{attribute 'linkalways'} 
{attribute 'no_explicit_call' := 'This FB is a CLASS and must be accessed using methods or properties'}
{attribute 'enable_dynamic_creation'}
FUNCTION_BLOCK _ETcVnSta EXTENDS EnumDatatypeBase
VAR
	localData : ETcVnSta;
	activeData : REFERENCE TO ETcVnSta;
	enumBaseDatatype : _UDINT(localData);
END_VAR

METHOD PRIVATE AddLocalEnumeration
VAR_INPUT
	Enumeration : T_MAXSTRING;
	Value : ETcVnSta;
END_VAR
AddEnumeration(Enumeration, Value);
END_METHOD

PROPERTY PUBLIC Address : PVOID
GET
Address := ADR(activeData);
END_GET
END_PROPERTY

METHOD PUBLIC ClearReference
VAR_INPUT
END_VAR
activeData REF= localData;
SetBaseDatatypeReference();
END_METHOD

METHOD PUBLIC Clone : I_Datatype
VAR
    pClone : POINTER TO _ETcVnSta;
END_VAR
pClone := __NEW(_ETcVnSta(InitialValue := Value));
Clone := pClone^;
END_METHOD

METHOD FB_init : BOOL
VAR_INPUT
	bInitRetains : BOOL; // if TRUE, the retain variables are initialized (warm start / cold start)
	bInCopyCode : BOOL;  // if TRUE, the instance afterwards gets moved into the copy code (online change)
	InitialValue : ETcVnSta;
END_VAR
localData := InitialValue;
AddBaseDatatype(enumBaseDatatype);
ClearReference();

AddLocalEnumeration('TCVN_STA_CLASSIFIER', ETcVnSta.TCVN_STA_CLASSIFIER);
AddLocalEnumeration('TCVN_STA_NOVELTY_DETECTOR', ETcVnSta.TCVN_STA_NOVELTY_DETECTOR);
AddLocalEnumeration('TCVN_STA_REGRESSOR', ETcVnSta.TCVN_STA_REGRESSOR);
AddLocalEnumeration('TCVN_STA_CLUSTERER', ETcVnSta.TCVN_STA_CLUSTERER);
END_METHOD

PROPERTY PUBLIC Identifier : T_MAXSTRING
GET
Identifier := 'ETcVnSta';
END_GET
END_PROPERTY

METHOD IsEnumeratorValueEqual : BOOL
VAR_INPUT
	Enumerator : I_KeyValueForwardEnumerator;
END_VAR
VAR
	storedValue : ETcVnSta;
END_VAR
IF NOT Enumerator.TryGet(storedValue) THEN
	RETURN;
END_IF

IsEnumeratorValueEqual := storedValue = activeData;
END_METHOD

METHOD PUBLIC MakeReferenceTo
VAR_INPUT
	ReferenceTarget : REFERENCE TO ETcVnSta;
END_VAR
activeData REF= ReferenceTarget;
SetBaseDatatypeReference();
END_METHOD

METHOD PROTECTED SetBaseDatatypeReference
VAR_INPUT
END_VAR
enumBaseDatatype.MakeReferenceTo(activeData);
END_METHOD

PROPERTY PUBLIC Size : UDINT
GET
Size := SIZEOF(activeData);
END_GET
END_PROPERTY

METHOD TryMakeReferenceTo : BOOL
VAR_INPUT
	Target : I_Datatype;
END_VAR
VAR
	pTargetData : POINTER TO ETcVnSta;
END_VAR
IF NOT IsEquivalentTo(Target) THEN
	RETURN;
END_IF

pTargetData := Target.Address;
activeData REF= pTargetData^;
SetBaseDatatypeReference();
TryMakeReferenceTo := TRUE;
END_METHOD

PROPERTY PUBLIC Value : ETcVnSta
GET
Value := activeData;
END_GET
SET
activeData := Value;
END_SET
END_PROPERTY

END_FUNCTION_BLOCK

(* stored: Version 1.1.0.1, ProductVersion 3.1.4024.13
   POU _ETcVnSta: Id {c6d70743-efbf-0625-1f69-70a08d218452}, SpecialFunc None
   Folder Core: Id {fbaa7d0f-cdf5-0dcd-30b6-0d5b45cef7cf}
   Folder Protected: Id {b4c42a9e-a3cf-0b64-05b7-09c25365ad76}
   Folder Customize: Id {e4b0e45f-ca16-043a-06ab-a132a95ea17d}
   Folder Constructor: Id {7af30cef-2414-0bd7-2350-14cd9528e980}
   Folder Private: Id {92c495f7-210f-0d8c-3f94-c9c292f7138d}
   Folder Protected: Id {d9b48cf6-f1d5-08ad-058f-d2a593b71f4e}
   Method AddLocalEnumeration: Id {fcdeac0a-2d6b-047b-1989-4e63b6a88972}
   Property Address: Id {9e5ee803-a270-0df2-066e-94ab8557abbf}
   Get Get: Id {56d1f39d-dca2-039b-29df-638efe179f82}
   Method ClearReference: Id {c5e75ae4-c578-07dc-1248-b0450194b1f9}
   Method Clone: Id {05af1d0b-ec02-070c-2db8-e12773cf7222}
   Method FB_init: Id {f4d1e336-385c-0a0c-14d1-ce0624d1ea6a}
   Property Identifier: Id {4e408104-a2c8-01a6-07cb-c3ad453bd48f}
   Get Get: Id {148bff92-fe22-098d-0888-135635ba6fd0}
   Method IsEnumeratorValueEqual: Id {9e9f0728-83d7-06f6-0a74-f85a0560b134}
   Method MakeReferenceTo: Id {87014744-46ff-061c-3f42-809719d12fbd}
   Method SetBaseDatatypeReference: Id {9ab2c472-8fc1-01a7-0bee-b106ae014aae}
   Property Size: Id {de1f5938-5fa8-050d-2dd0-983e7774e433}
   Get Get: Id {e0f6e7f4-a653-0561-15a7-02c197cde581}
   Method TryMakeReferenceTo: Id {47e6b736-8937-0998-3fb4-a92648bf9eb0}
   Property Value: Id {80b68b02-93a0-0efd-2a24-72fad2b664d3}
   Get Get: Id {7bc9be0e-0b94-0f3a-0465-e48227d9828b}
   Set Set: Id {d14d99b3-f306-0c2a-01a9-d6424e0aa929} *)
